{attribute 'GeneratedUsingTerminal: AMP8000-0030-0103-0103'}
{attribute addProperty BoxType "AMP8000-0030-0103-0103"}
{attribute addProperty Id "Ch_A_ControlwordAT %Q*UINT2"}
{attribute addProperty CRC "2845499694"}
{attribute addProperty Size "2"}
TYPE Ch_A_AxisMain_Outputs_A99AE12E EXTENDS OutputBase_10CEE7DE :
STRUCT
	{attribute addProperty Name "Ch_A_Controlword"}
	Ch_A_Controlword AT %Q* : UINT;
END_STRUCT
END_TYPE

(* stored: Version 1.2.0.0, ProductVersion 3.1.4024.11
   DUT Ch_A_AxisMain_Outputs_A99AE12E: Id {c81d4422-9f65-4cd0-999c-de026e978575} *)
